Universal Robots PolyScope program: adaptr_grip.urp

Program adaptr_grip (installation=default directory=/programs/Demos/adaptiveGrip createdIn=5.13.1 lastSavedIn=5.15.1 robotSerialNumber=20245500285)
Calibrated DH parameters: a=[0.000097, -0.210459, -0.026602, 0.000137, 0.000078, 0]; d=[0.162601, 254.180657, -54.076236, -199.970743, 0.099615, 0.099684]; alpha=[1.569796, -0.001455, 0.001957, 1.570525, -1.571561, 0]; deltaTheta=[0, -1.053331, 8.839472, -1.50296, 0.000002, 0]
InitVariablesNode
Robot Program (runOnlyOnce=true)
  Script: usb = rpc_factory("xmlrpc","http://192.168.1.7:9120/RPC2")
  Script: usb.open()
  SuppressedNode
    Wait Sleep waitTime=2
  SuppressedNode
    Script: usb.close()
  SuppressedNode
    Script: usb.adaptive_close()
